// TIA Portal V15.1 export
// export: Created 2024-05-17T05:38:21.638085Z, ExportSetting WithDefaults, DisplayName Totally Integrated Automation Portal, DisplayVersion V15.1 Update 5, DisplayName TIA Portal Openness, DisplayVersion V15.1 Update 5, DisplayName SINAMICS Startdrive Advanced, DisplayVersion V15.1, DisplayName G130, G150, S120, S150, SINAMICS MV, S210, DisplayVersion V15.1, DisplayName G110M, G120, G120C, G120D, G120P, DisplayVersion V15.1, DisplayName STEP 7 Professional, DisplayVersion V15.1 Update 5, DisplayName STEP 7 Safety, DisplayVersion V15.1, DisplayName WinCC Professional, DisplayVersion V15.1 Update 5, DisplayName SIMATIC Visualization Architect, DisplayVersion V15.1
DATA_BLOCK "_209230ZS01AEAK"   // DB421
{ S7_Optimized_Access := 'FALSE' }
AUTHOR : VCC
VERSION : 0.1
// stored: AutoNumber false, DBAccessibleFromOPCUA true, IsOnlyStoredInLoadMemory false, IsWriteProtectedInAS false
   VAR RETAIN
      AB_AK01E1QM14 { ExternalAccessible := 'False'; ExternalVisible := 'False'; ExternalWritable := 'False'} : Bool;   // 400VAC - Overload protection MoviFit chain Mode Zone 230
      AA_AE01E3FS13_CH1 { ExternalAccessible := 'False'; ExternalVisible := 'False'; ExternalWritable := 'False'} : Bool;   // 24VDC Fuse - ModeZone230 - Switch / Busnode 230AX01 & 230AS10
      AC_AE01E3FS13_CH2 { ExternalAccessible := 'False'; ExternalVisible := 'False'; ExternalWritable := 'False'} : Bool;   // 24VDC Fuse - ModeZone230 - RFID Reader
      AD_AE01E3FS13_CH1 { ExternalAccessible := 'False'; ExternalVisible := 'False'; ExternalWritable := 'False'} : Bool;   // 24VDC Fuse - ModeZone230 - Switch / Busnode 230AX01 & 230AS10
      AD_AE01E3FS13_CH2 { ExternalAccessible := 'False'; ExternalVisible := 'False'; ExternalWritable := 'False'} : Bool;   // 24VDC Fuse - ModeZone230 - RFID Reader
      AA_AK02E3FS300_CH1 { ExternalAccessible := 'False'; ExternalVisible := 'False'; ExternalWritable := 'False'} : Bool;   // 24VDC Fuse - ModeZone 230 - DI/DO 230AX01 & 230AS10
      AA_AK02E3FS300_CH2 { ExternalAccessible := 'False'; ExternalVisible := 'False'; ExternalWritable := 'False'} : Bool;   // 24VDC Fuse - ModeZone 230 - F-DI/F-DO 230AX01 & 230AS10
      AA_AK02E3FS301_CH1 { ExternalAccessible := 'False'; ExternalVisible := 'False'; ExternalWritable := 'False'} : Bool;   // 24VDC Fuse - ModeZone 230 - Doorlock
      AA_AK02E3FS301_CH2 { ExternalAccessible := 'False'; ExternalVisible := 'False'; ExternalWritable := 'False'} : Bool;   // 24VDC Fuse - ModeZone 230 - Lightcurtain
      AB_AK02E3FS302_CH1 { ExternalAccessible := 'False'; ExternalVisible := 'False'; ExternalWritable := 'False'} : Bool;   // 24VDC Fuse - ModeZone 230 - Movifit Chain 1
      AD_AK02E3FS300_CH1 { ExternalAccessible := 'False'; ExternalVisible := 'False'; ExternalWritable := 'False'} : Bool;   // 24VDC Fuse - ModeZone 230 - DI/DO 230AX01 & 230AS10
      AD_AK02E3FS300_CH2 { ExternalAccessible := 'False'; ExternalVisible := 'False'; ExternalWritable := 'False'} : Bool;   // 24VDC Fuse - ModeZone 230 - F-DI/F-DO 230AX01 & 230AS10
      AD_AK02E3FS301_CH1 { ExternalAccessible := 'False'; ExternalVisible := 'False'; ExternalWritable := 'False'} : Bool;   // 24VDC Fuse - ModeZone 230 - Doorlock
      AD_AK02E3FS301_CH2 { ExternalAccessible := 'False'; ExternalVisible := 'False'; ExternalWritable := 'False'} : Bool;   // 24VDC Fuse - ModeZone 230 - Lightcurtain
      AD_AK02E3FS302_CH1 { ExternalAccessible := 'False'; ExternalVisible := 'False'; ExternalWritable := 'False'} : Bool;   // 24VDC Fuse - ModeZone 230 - Movifit Chain 1
      AK01E1QM14AlarmABCondition { ExternalAccessible := 'False'; ExternalVisible := 'False'; ExternalWritable := 'False'} : Bool;   // Alarm AB condition
      AE01E3FS13_CH1AlarmABCondition { ExternalAccessible := 'False'; ExternalVisible := 'False'; ExternalWritable := 'False'} : Bool;   // Alarm AB condition
      AK02E3FS300_CH1AlarmABCondition { ExternalAccessible := 'False'; ExternalVisible := 'False'; ExternalWritable := 'False'} : Bool;   // Alarm AB condition
      AK02E3FS300_CH2AlarmABCondition { ExternalAccessible := 'False'; ExternalVisible := 'False'; ExternalWritable := 'False'} : Bool;   // Alarm AB condition
      AK02E3FS301_CH1AlarmABCondition { ExternalAccessible := 'False'; ExternalVisible := 'False'; ExternalWritable := 'False'} : Bool;   // Alarm AB condition
      AK02E3FS301_CH2AlarmABCondition { ExternalAccessible := 'False'; ExternalVisible := 'False'; ExternalWritable := 'False'} : Bool;   // Alarm AB condition
      AK02E3FS302_CH1AlarmABCondition { ExternalAccessible := 'False'; ExternalVisible := 'False'; ExternalWritable := 'False'} : Bool;   // Alarm AB condition
      H_209000AK01E1QM14IAnim : Word;   // HMI Animation of the icon
      H_209000AE01E3FS13_CH1IAnim : Word;   // HMI Animation of the icon
      H_209000AE01E3FS13_CH2IAnim : Word;   // HMI Animation of the icon
      H_209000AK02E3FS300_CH1IAnim : Word;   // HMI Animation of the icon
      H_209000AK02E3FS300_CH2IAnim : Word;   // HMI Animation of the icon
      H_209000AK02E3FS301_CH1IAnim : Word;   // HMI Animation of the icon
      H_209000AK02E3FS301_CH2IAnim : Word;   // HMI Animation of the icon
      H_209000AK02E3FS302_CH1IAnim : Word;   // HMI Animation of the icon
      H_209000AK02E3FS302_CH2IAnim : Word;   // HMI Animation of the icon
      H_209000AK02E3FS303_CH1IAnim : Word;   // HMI Animation of the icon
      H_209000AK02E3FS303_CH2IAnim : Word;   // HMI Animation of the icon
      H_DBnr : Int;   // DB number
      H_Anim : Word;   // Animation
      AlarmA { ExternalAccessible := 'False'; ExternalVisible := 'False'; ExternalWritable := 'False'} : Bool;   // Alarm A
      AlarmB { ExternalAccessible := 'False'; ExternalVisible := 'False'; ExternalWritable := 'False'} : Bool;   // Alarm B
      AlarmC { ExternalAccessible := 'False'; ExternalVisible := 'False'; ExternalWritable := 'False'} : Bool;   // Alarm C
      AlarmD { ExternalAccessible := 'False'; ExternalVisible := 'False'; ExternalWritable := 'False'} : Bool;   // Alarm D
      AlarmABCondition { ExternalAccessible := 'False'; ExternalVisible := 'False'; ExternalWritable := 'False'} : Bool;   // Alarm AB condition
   END_VAR
BEGIN
END_DATA_BLOCK
